(* CODESYS project TrafficLight.project

Project tree, tasks and I/O mapping:
  Device : Elmo Platinum Maestro, Elmo Motion Control, version 1.0.0.2
    application Application
      libraries: Standard, * (System); VisuDialogs, * (System)
      task MainTask (cyclic, interval t#20ms, priority 1) calls PLC_PRG
      task VISU_TASK (cyclic, interval 100 ms, priority 31) calls VisuElems.Visu_Prg
      program PLC_PRG [ST]
      visualisation Visualization
      Structure/
        data type stCarX
        data type stCarY
      function block fbModeSwitch [ST]
      function fTimetoString [ST]
      function block fbGreenTimeCondition [ST]
      function block fbYellowTimeCondition [ST]
      function block fbClearTimeCondition [ST]
      function block fbFrontandBackCar [ST]
    Elmo_Master_Device : Elmo Master Device, Elmo, version 1.0.0.2
  libraries: VisuSymbols, 3.5.10.0 (System)
  text list GlobalTextList
*)

// Device/Application/Structure/stCarX
TYPE stCarX :
STRUCT
	iMove_x: INT;
	//iBase_x: ARRAY[1..5] OF INT := [243,195,157,113,69];
	//iBase_x: ARRAY[1..5] OF INT;
END_STRUCT
END_TYPE

// Device/Application/Structure/stCarY
TYPE stCarY :
STRUCT
	iMove_y: INT;
	//iBase_y: ARRAY[1..5] OF INT;
END_STRUCT
END_TYPE

// Device/Application/PLC_PRG
PROGRAM PLC_PRG
VAR CONSTANT
	c_dwRoadColor : DWORD := 16#88888888;
	c_dwLaneColor: DWORD := 16#FFFFFF00;
	c_dwTLbg: DWORD := 16#88000000;
END_VAR
VAR
	xPush: BOOL;
	tonTimer1: ton;
	tonTimer2: ton;
	tonTimer3: ton;
	xStart1: BOOL;
	xStart2: BOOL;
	xStart3: BOOL;
	uiTrafficSig: UINT:=0;
	
	xGreen1 : BOOL;
	xYellow1 : BOOL;
	xRed1 : BOOL;
	xRed2 : BOOL;
	xYellow2 : BOOL;
	xGreen2 : BOOL;
	tTimer1: TIME := T#7000MS;
	tTimer2: TIME := T#5000MS;
	tTimer3: TIME := T#4000MS;
	
	tSTime1: STRING := 'T#7s';
	tSTime2: STRING := 'T#5s';
	tSTime3: STRING := 'T#4s';
	
	tSeTime1: STRING := 'T#7s';
	tSeTime2: STRING := 'T#5s';
	tSeTime3: STRING := 'T#4s';
	tRed : STRING;
	
	tEditTime1 : TIME := T#7000MS;
	tEditTime2 : TIME := T#5000MS;
	tEditTime3 : TIME := T#4000MS;
	sEditTime1 : STRING;
	sEditTime2 : STRING;
	sEditTime3 : STRING;
	
	stCarX: ARRAY [1..5] OF stCarX;
	uiLoop: UINT;
	
	iBase_x : ARRAY[1..5] OF INT := [250,200,150,100,50];
		
	stCarY: ARRAY [1..5] OF stCarY;
	uiLoop2: UINT;
	iBase_y : ARRAY[1..5] OF INT := [450,500,550,600,650];
	
	iMoveUser1X: INT;
	iMoveUser1Y: INT;
	iMoveUser2X: INT;
	iMoveUser2Y: INT;
	iMoveUser1Z: INT;
	iMoveUser2Z: INT;
	
	iCurrent: INT;
	iCurrent2: INT;
	iForward: INT;
	iForward2: INT;
	iBack: INT;
	iBack2: INT;
    sMode: STRING;
	iTemp: INT;
	iTemp2: INT;
	iStart: INT;
	iStart2: INT;
	
	fbMode : fbModeSwitch;
	fbGreenTime: fbGreenTimeCondition;
	fbYellowTime: fbYellowTimeCondition;
	fbClearTime: fbClearTimeCondition;
	fbFrontBack: fbFrontandBackCar;
END_VAR

//Mode Switch
fbMode(ix_Push := xPush,os_Mode => sMode);

//Time Edit
tSTime1 := fTimetoString(it_Time := tTimer1);
tSTime2 := fTimetoString(it_Time := tTimer2);
tSTime3 := fTimetoString(it_Time := tTimer3);
tSeTime1 := fTimetoString(it_Time := tEditTime1);
tSeTime2 := fTimetoString(it_Time := tEditTime2);
tSeTime3 := fTimetoString(it_Time := tEditTime3);

//Green Time Edit Conditions
fbGreenTime(it_EditTime1 := tEditTime1 ,it_Timer2 := tTimer2 ,it_Timer3 := tTimer3 ,ot_timer1 => tTimer1 ,os_EditTime1 => sEditTime1);
//Yellow Time Edit Conditions
fbYellowTime(it_EditTime2 := tEditTime2 ,it_EditTime1 := tEditTime1 ,it_EditTime3 := tEditTime3 ,ot_timer2 => tTimer2 ,os_EditTime2 => sEditTime2);
//Clear Time Edit Conditions
fbClearTime(it_EditTime3 := tEditTime3 ,it_EditTime1 := tEditTime1 ,it_EditTime2 := tEditTime2 ,ot_timer3 => tTimer3 ,os_EditTime3 => sEditTime3);

//Traffic Light Sequence
CASE uiTrafficSig OF
	0:
	     xRed1 := FALSE;
	     xGreen1 := TRUE;
	     xRed2 := TRUE;
	     tonTimer1(IN := xStart1, PT := tTimer1);
	     xStart1 := TRUE;
	     IF tonTimer1.Q = TRUE THEN
		   xStart1 := FALSE;
		   xGreen1 := FALSE;
		   uiTrafficSig := 10;
	     END_IF
	10:
	   tonTimer2(IN := xStart2, PT := tTimer2);
	   xStart2 := TRUE;
	   xYellow1 := TRUE;
	   IF tonTimer2.Q = TRUE THEN
		   xStart2 := FALSE;
		   //xYellow1 := FALSE;
		   uiTrafficSig := 20;
	   END_IF
	20:
	   tonTimer3(IN := xStart3, PT := tTimer3);
	   xStart3 := TRUE;
	   xYellow1 := FALSE;
	   xRed1 := TRUE;
	   IF tonTimer3.Q = TRUE THEN
		   xStart3 := FALSE;
		   IF xPush = TRUE THEN
			   uiTrafficSig := 60;
		   ELSE
			   uiTrafficSig := 30;
		   END_IF
	   END_IF
	30:
	       xRed2 := FALSE;
	       xGreen2 := TRUE;
	       tonTimer1(IN := xStart1, PT := tTimer1);
	       xStart1 := TRUE;
	       IF tonTimer1.Q = TRUE THEN
			   xStart1 := FALSE;
			   xGreen2 := FALSE;
			   uiTrafficSig := 40;
	       END_IF
	40:
	   xYellow2 := TRUE;
	   tonTimer2(IN := xStart2, PT := tTimer2);
	   xStart2 := TRUE;
	   IF tonTimer2.Q = TRUE THEN
		   xStart2 := FALSE;
		   //xYellow2 := FALSE;
		   uiTrafficSig := 50;
	   END_IF
	50:
	   xYellow2 := FALSE;
	   xRed2 := TRUE;
	   tonTimer3(IN := xStart3, PT := tTimer3);
	   xStart3 := TRUE;
	   IF tonTimer3.Q = TRUE THEN
		   xStart3 := FALSE;
		   IF xPush = TRUE THEN
			   uiTrafficSig := 60;
		   ELSE
			   uiTrafficSig := 0;
		   END_IF
	   END_IF
	60:
	IF xPush = TRUE THEN
	   xRed1 := TRUE;
	   xRed2 := TRUE;
	   xYellow1 := FALSE;
	   xYellow2 := FALSE;
	   xGreen1 := FALSE;
	   xGreen2 := FALSE;
	ELSE
		uiTrafficSig := 0;
	END_IF
END_CASE

//Red Time Total
tRed := fTimetoString(it_Time := tTimer1 + tTimer2 + tTimer3);

FOR uiLoop:=1 TO 5 BY 1 DO
	iCurrent := iBase_x[uiLoop] + stCarX[uiLoop].iMove_x;
	
    IF xGreen1 = TRUE OR xYellow1 = TRUE THEN
		iTemp := 0;
		FOR uiLoop2:=1 TO 5 BY 1 DO
			//knowing front and back cars of each
			fbFrontBack(iui_Loop:=uiLoop,ii_Base_x:=iBase_x,stCarX:=stCarX,oi_Forward => iForward, oi_Back => iBack);
			
			//condition 1 for stopping at green signal if any opposite cars are seen at intersection
			IF iBase_y[uiLoop2] + stCarY[uiLoop2].iMove_y < 450 AND iBase_y[uiLoop2] + stCarY[uiLoop2].iMove_y > 175 THEN
				stCarX[uiLoop].iMove_x := stCarX[uiLoop].iMove_x +0;
				iTemp := 0;
			ELSE
					IF iBase_y[uiLoop2] + stCarY[uiLoop2].iMove_y > 450 OR iBase_y[uiLoop2] + stCarY[uiLoop2].iMove_y < 175 THEN
						iTemp := iTemp + 1;
					END_IF
				
			END_IF
		END_FOR
		
		//condition 2 for stopping at green signal if any opposite cars are seen at intersection
		IF iCurrent >= 425 AND iCurrent < 450 AND iTemp < 5 THEN
			stCarX[uiLoop].iMove_x := stCarX[uiLoop].iMove_x +0;
			IF uiLoop = 5 THEN
					stCarX[1].iMove_x := stCarX[1].iMove_x + 0;
			ELSE
					stCarX[uiLoop + 1].iMove_x := stCarX[uiLoop + 1].iMove_x + 0;
			END_IF
		END_IF
		
		//Condition for car movement at green signal and also condition for reverse
		IF (iTemp >= 4 OR (iCurrent < 425 AND iForward - iCurrent > 50 AND iForward > iCurrent) OR (iCurrent > 450) OR (iCurrent < 425 AND iCurrent - iForward > 50 AND iCurrent > iForward)) THEN
			IF stCarX[uiLoop].iMove_x <= -500 THEN
				IF iStart >= 5 THEN
					stCarX[uiLoop].iMove_x := stCarX[uiLoop].iMove_x +1;
				ELSE
					stCarX[uiLoop].iMove_x := stCarX[uiLoop].iMove_x +0;
				END_IF
			ELSE
				stCarX[uiLoop].iMove_x := stCarX[uiLoop].iMove_x +1;
			END_IF
		END_IF
		
	ELSIF xRed1 = TRUE THEN
		iTemp:= 0;
		iCurrent := iBase_x[uiLoop] + stCarX[uiLoop].iMove_x;

		fbFrontBack(iui_Loop:=uiLoop,ii_Base_x:=iBase_x,stCarX:=stCarX,oi_Forward => iForward, oi_Back => iBack);
			//Movement Condition 1 and reverse condition during red light
			IF iCurrent < 425 AND iForward - iCurrent > 50 AND iForward > iCurrent THEN
				IF stCarX[uiLoop].iMove_x <= -500 THEN
				 IF iStart >= 5 THEN
					stCarX[uiLoop].iMove_x := stCarX[uiLoop].iMove_x +1;
				 ELSE
					stCarX[uiLoop].iMove_x := stCarX[uiLoop].iMove_x +0;
				 END_IF
			  ELSE
				stCarX[uiLoop].iMove_x := stCarX[uiLoop].iMove_x +1;
			END_IF
				
			//Movement Condition 2 and reverse condition during red light
			ELSIF iCurrent < 425 AND iForward < 425 AND iCurrent - iForward > 50 THEN
				IF stCarX[uiLoop].iMove_x <= -500 THEN
				 IF iStart >= 5 THEN
					stCarX[uiLoop].iMove_x := stCarX[uiLoop].iMove_x +1;
				 ELSE
					stCarX[uiLoop].iMove_x := stCarX[uiLoop].iMove_x +0;
				 END_IF
			   ELSE
				stCarX[uiLoop].iMove_x := stCarX[uiLoop].iMove_x +1;
			  END_IF
			
          //Stop Condition 1	
		  ELSIF iCurrent < 425 THEN
			  stCarX[uiLoop].iMove_x := stCarX[uiLoop].iMove_x + 0;
		  //Intersection Speeding Condition
		  ELSIF iCurrent > 425 AND iCurrent < 800 THEN
			  stCarX[uiLoop].iMove_x := stCarX[uiLoop].iMove_x + 5;
			
          //Movement Condition 3	
		  ELSIF iCurrent >= 800 THEN
			  stCarX[uiLoop].iMove_x := stCarX[uiLoop].iMove_x + 5;
			  
			END_IF
			
	END_IF
		
	//Condition at end
	IF iBase_x[uiLoop] + stCarX[uiLoop].iMove_x >= 1900 THEN
		fbFrontBack(iui_Loop:=uiLoop,ii_Base_x:=iBase_x,stCarX:=stCarX,oi_Forward => iForward, oi_Back => iBack);
		
		IF(iStart >= 5)THEN
			iStart := 0;
		END_IF
		stCarX[uiLoop].iMove_x := -500;
		iStart := iStart + 1;
    END_IF
	
END_FOR

FOR uiLoop2:=1 TO 5 BY 1 DO
	
	iCurrent2 := iBase_y[uiLoop2] + stCarY[uiLoop2].iMove_y;
	
	IF xGreen2 = TRUE OR xYellow2 = TRUE THEN
		iTemp2 := 0;
		FOR uiLoop:=1 TO 5 BY 1 DO
			IF uiLoop2 = 1 THEN
				iForward2 := iBase_y[5] + stCarY[5].iMove_y;
			    iBack2 := iBase_y[uiLoop2 + 1] + stCarY[uiLoop2 + 1].iMove_y;
			ELSIF uiLoop2 = 5 THEN
				iForward2 := iBase_y[uiLoop2 - 1] + stCarY[uiLoop2 - 1].iMove_y;
			    iBack2 := iBase_y[1] + stCarY[1].iMove_y;
			ELSE
				iForward2 := iBase_y[uiLoop2 - 1] + stCarY[uiLoop2 - 1].iMove_y;
			    iBack2 := iBase_y[uiLoop2 + 1] + stCarY[uiLoop2 + 1].iMove_y;
			END_IF
			//condition 1 for stopping at green signal if any opposite cars are seen at intersection
			IF iBase_x[uiLoop] + stCarX[uiLoop].iMove_x > 425 AND iBase_x[uiLoop] + stCarX[uiLoop].iMove_x < 800 THEN
				stCarX[uiLoop].iMove_x := stCarX[uiLoop].iMove_x +0;
				iTemp2 := 0;
			ELSE
					IF iBase_x[uiLoop] + stCarX[uiLoop].iMove_x < 425 OR iBase_x[uiLoop] + stCarX[uiLoop].iMove_x > 800 THEN
						iTemp2 := iTemp2 + 1;
					END_IF
				
			END_IF
		END_FOR
		
		//condition 2 for stopping at green signal if any opposite cars are seen at intersection
		IF iCurrent2 <= 450 AND iCurrent2 > 425 AND iTemp2 < 5 THEN
			stCarY[uiLoop2].iMove_y := stCarY[uiLoop2].iMove_y +0;
			IF uiLoop2 = 5 THEN
					stCarY[1].iMove_y := stCarY[1].iMove_y + 0;
			ELSE
					stCarY[uiLoop2 + 1].iMove_y := stCarY[uiLoop2 + 1].iMove_y + 0;
			END_IF
		END_IF
		//Condition for car movement at green signal and also condition for reverse
		IF iTemp2 >= 4 OR (iCurrent2 > 450 AND iCurrent2 - iForward2 > 50 AND iForward2 < iCurrent2) OR (iCurrent2 < 425) OR (iCurrent2 > 450 AND iForward2 - iCurrent2 > 50 AND iCurrent2 < iForward2)THEN
			IF stCarY[uiLoop2].iMove_y >= 1050 THEN
				IF iStart2 >= 5 THEN
					stCarY[uiLoop2].iMove_y := stCarY[uiLoop2].iMove_y -1;
				ELSE
					stCarY[uiLoop2].iMove_y := stCarY[uiLoop2].iMove_y +0;
				END_IF
			ELSE
				stCarY[uiLoop2].iMove_y := stCarY[uiLoop2].iMove_y -1;
			END_IF
		END_IF
		
		
	ELSIF xRed2 = TRUE THEN
		iCurrent2 := iBase_y[uiLoop2] + stCarY[uiLoop2].iMove_y;
		iTemp2 := 0;
		
			IF uiLoop2 = 1 THEN
				iForward2 := iBase_y[5] + stCarY[5].iMove_y;
			    iBack2 := iBase_y[uiLoop2 + 1] + stCarY[uiLoop2 + 1].iMove_y;
			ELSIF uiLoop2 = 5 THEN
				iForward2 := iBase_y[uiLoop2 - 1] + stCarY[uiLoop2 - 1].iMove_y;
			    iBack2 := iBase_y[1] + stCarY[1].iMove_y;
			ELSE
				iForward2 := iBase_y[uiLoop2 - 1] + stCarY[uiLoop2 - 1].iMove_y;
			    iBack2 := iBase_y[uiLoop2 + 1] + stCarY[uiLoop2 + 1].iMove_y;
			END_IF
			//Movement Condition 1 and reverse condition during red light
			IF iCurrent2 > 450 AND  iCurrent2 - iForward2 > 50 AND iForward2 < iCurrent2 THEN
				IF stCarY[uiLoop2].iMove_y >= 1050 THEN
				 IF iStart2 >= 5 THEN
					stCarY[uiLoop2].iMove_y := stCarY[uiLoop2].iMove_y -1;
				 ELSE
					stCarY[uiLoop2].iMove_y := stCarY[uiLoop2].iMove_y +0;
				 END_IF
			   ELSE
				stCarY[uiLoop2].iMove_y := stCarY[uiLoop2].iMove_y -1;
			   END_IF
			   //Movement Condition 2 and reverse condition during red light
			ELSIF iCurrent2 > 450 AND iForward2 > 450 AND  iForward2 - iCurrent2 > 50 THEN
				IF stCarY[uiLoop2].iMove_y >= 1050 THEN
				 IF iStart2 >= 5 THEN
					stCarY[uiLoop2].iMove_y := stCarY[uiLoop2].iMove_y -1;
				 ELSE
					stCarY[uiLoop2].iMove_y := stCarY[uiLoop2].iMove_y +0;
				 END_IF
			   ELSE
				stCarY[uiLoop2].iMove_y := stCarY[uiLoop2].iMove_y -1;
			   END_IF
			   //Stop Condition 1
			ELSIF iCurrent2 > 450 THEN
			  stCarY[uiLoop2].iMove_y := stCarY[uiLoop2].iMove_y + 0;
			  //Intersection Speeding Condition
			ELSIF iCurrent2 < 450 AND iCurrent2 > 175 THEN
			    stCarY[uiLoop2].iMove_Y := stCarY[uiLoop2].iMove_y - 5;
				
				//Movement Condition 3
		    ELSIF iCurrent2 <= 175 THEN
			  stCarY[uiLoop2].iMove_y := stCarY[uiLoop2].iMove_y - 5;
			  
			END_IF
			
	END_IF
		
		//Condition at end
	IF iBase_y[uiLoop2] + stCarY[uiLoop2].iMove_y <= -100 THEN
		IF uiLoop2 = 1 THEN
				iForward2 := iBase_y[5] + stCarY[5].iMove_y;
			    iBack2 := iBase_y[uiLoop2 + 1] + stCarY[uiLoop2 + 1].iMove_y;
		ELSIF uiLoop = 5 THEN
				iForward2 := iBase_y[uiLoop2 - 1] + stCarY[uiLoop2 - 1].iMove_y;
			    iBack2 := iBase_y[1] + stCarY[1].iMove_y;
		ELSE
				iForward2 := iBase_y[uiLoop2 - 1] + stCarY[uiLoop2 - 1].iMove_y;
			    iBack2 := iBase_y[uiLoop2 + 1] + stCarY[uiLoop2 + 1].iMove_y;
		END_IF
			IF(iStart2 >= 5)THEN
			  iStart2 := 0;
		    END_IF
		    stCarY[uiLoop2].iMove_y := 1050;
		    iStart2 := iStart2 + 1;
    END_IF
	
END_FOR

//People Movement at crossing
CASE iMoveUser1Z OF
	0:
	   IF xGreen1 = TRUE THEN
		   iMoveUser1X := iMoveUser1X + 5;
	       IF iMoveUser1X = 250 THEN
	         iMoveUser1Z:= 250;
	       END_IF
	   END_IF
	   
	250:
	   IF xGreen2 = TRUE THEN
		   iMoveUser1Y := iMoveUser1Y - 5;
		   IF iMoveUser1Y = -175 THEN
	         iMoveUser1Z:= 500;
	       END_IF
	   END_IF
	   
	500:
	   IF xGreen1 = TRUE THEN
		   iMoveUser1X := iMoveUser1X - 5;
	       IF iMoveUser1X = 0 THEN
	         iMoveUser1Z:= 750;
	       END_IF
	   END_IF
	   
	 750:
	   IF xGreen2 = TRUE THEN
		   iMoveUser1Y := iMoveUser1Y + 5;
		   IF iMoveUser1Y = 0 THEN
	         iMoveUser1Z:= 0;
	       END_IF
	   END_IF
		
END_CASE


CASE iMoveUser2Z OF
	0:
	   IF xGreen1 = TRUE THEN
		   iMoveUser2X := iMoveUser2X - 5;
	       IF iMoveUser2X = -225 THEN
	         iMoveUser2Z:= 250;
	       END_IF
	   END_IF
	   
	250:
	   IF xGreen2 = TRUE THEN
		   iMoveUser2Y := iMoveUser2Y + 5;
		   IF iMoveUser2Y = 175 THEN
	         iMoveUser2Z:= 500;
	       END_IF
	   END_IF
	   
	500:
	   IF xGreen1 = TRUE THEN
		   iMoveUser2X := iMoveUser2X + 5;
	       IF iMoveUser2X = 0 THEN
	         iMoveUser2Z:= 750;
	       END_IF
	   END_IF
	   
	 750:
	   IF xGreen2 = TRUE THEN
		   iMoveUser2Y := iMoveUser2Y - 5;
		   IF iMoveUser2Y = 0 THEN
	         iMoveUser2Z:= 0;
	       END_IF
	   END_IF
		
END_CASE

END_PROGRAM

// Device/Application/fTimetoString
FUNCTION fTimetoString : STRING
VAR_INPUT
	it_Time: TIME;
END_VAR
VAR
END_VAR

fTimetoString := TIME_TO_STRING(it_Time);

END_FUNCTION

// Device/Application/fbModeSwitch
FUNCTION_BLOCK fbModeSwitch
VAR_INPUT
	ix_Push: BOOL;
END_VAR
VAR_OUTPUT
	os_Mode: STRING;
END_VAR
VAR
END_VAR

IF ix_Push = TRUE THEN
	os_Mode := 'STOP';
ELSE
	os_Mode := 'AUTO';
END_IF

END_FUNCTION_BLOCK

// Device/Application/fbGreenTimeCondition
FUNCTION_BLOCK fbGreenTimeCondition
VAR_INPUT
	it_EditTime1: TIME;
	it_Timer2: TIME;
	it_Timer3: TIME;
END_VAR
VAR_OUTPUT
	ot_Timer1: TIME;
	os_EditTime1: STRING;
END_VAR
VAR
END_VAR

IF it_EditTime1 >= T#7000MS AND it_EditTime1 > it_Timer2 AND it_EditTime1 > it_Timer3 AND it_EditTime1 <= T#30000MS THEN
			 ot_Timer1 := it_EditTime1;
			 os_EditTime1 := 'Valid';
ELSE
	os_EditTime1 := 'Invalid';
END_IF

END_FUNCTION_BLOCK

// Device/Application/fbYellowTimeCondition
FUNCTION_BLOCK fbYellowTimeCondition
VAR_INPUT
	it_EditTime2: TIME;
	it_EditTime1: TIME;
	it_EditTime3: TIME;
END_VAR
VAR_OUTPUT
	ot_Timer2: TIME;
	os_EditTime2: STRING;
END_VAR
VAR
END_VAR

IF it_EditTime2 >= T#5000MS AND it_EditTime2 < it_EditTime1 AND it_EditTime2 > it_EditTime3 AND it_EditTime2 <= T#28000MS THEN
			 ot_Timer2 := it_EditTime2;
			 os_EditTime2 := 'Valid';
ELSE
	os_EditTime2 := 'Invalid';
END_IF

END_FUNCTION_BLOCK

// Device/Application/fbClearTimeCondition
FUNCTION_BLOCK fbClearTimeCondition
VAR_INPUT
	it_EditTime3: TIME;
	it_EditTime1: TIME;
	it_EditTime2: TIME;
END_VAR
VAR_OUTPUT
	ot_Timer3: TIME;
	os_EditTime3: STRING;
END_VAR
VAR
END_VAR

IF it_EditTime3 >= T#4000MS AND it_EditTime3 < it_EditTime1 AND it_EditTime3 < it_EditTime2 AND it_EditTime3 <= T#27000MS THEN
			 ot_Timer3 := it_EditTime3;
			 os_EditTime3 := 'Valid';
ELSE
	os_EditTime3 := 'Invalid';
END_IF

END_FUNCTION_BLOCK

// Device/Application/fbFrontandBackCar
FUNCTION_BLOCK fbFrontandBackCar
VAR_INPUT
	iui_Loop: UINT;
	ii_Base_x : ARRAY[1..5] OF INT := [250,200,150,100,50];
	stCarX: ARRAY [1..5] OF stCarX;
END_VAR
VAR_OUTPUT
	oi_Forward: INT;
	oi_Back: INT;
END_VAR
VAR
END_VAR

IF iui_Loop = 1 THEN
		oi_Forward := ii_Base_x[5] + stCarX[5].iMove_x;
	    oi_Back := ii_Base_x[iui_Loop + 1] + stCarX[iui_Loop + 1].iMove_x;
ELSIF iui_Loop = 5 THEN
		oi_Forward := ii_Base_x[iui_Loop - 1] + stCarX[iui_Loop - 1].iMove_x;
		oi_Back := ii_Base_x[1] + stCarX[1].iMove_x;
ELSE
		oi_Forward := ii_Base_x[iui_Loop - 1] + stCarX[iui_Loop - 1].iMove_x;
	    oi_Back := ii_Base_x[iui_Loop + 1] + stCarX[iui_Loop + 1].iMove_x;
END_IF

END_FUNCTION_BLOCK

// Device/Application/Visualization
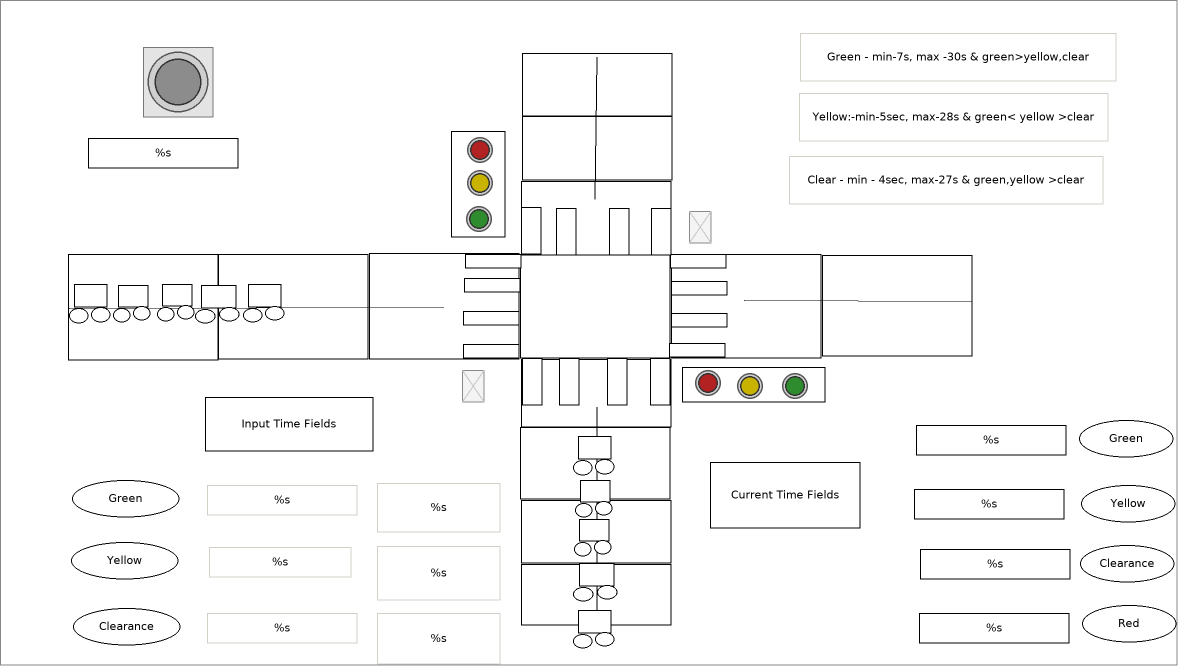
VISUALIZATION Visualization  // 1178x666
    Rectangle (68,254 150x106), colour variable: PLC_PRG.c_dwRoadColor
    Rectangle (218,254 150x105), colour variable: PLC_PRG.c_dwRoadColor
    Rectangle (369,253 150x106), colour variable: PLC_PRG.c_dwRoadColor
    Rectangle (520,254 150x104), colour variable: PLC_PRG.c_dwRoadColor
    Rectangle (671,254 150x104), colour variable: PLC_PRG.c_dwRoadColor
    Rectangle (822,255 150x101), colour variable: PLC_PRG.c_dwRoadColor
    Rectangle (521,181 150x74), colour variable: PLC_PRG.c_dwRoadColor
    Rectangle (522,116 150x64), colour variable: PLC_PRG.c_dwRoadColor
    Rectangle (522,53 150x63), colour variable: PLC_PRG.c_dwRoadColor
    Rectangle (521,359 150x68), colour variable: PLC_PRG.c_dwRoadColor
    Rectangle (520,427 150x72), colour variable: PLC_PRG.c_dwRoadColor
    Rectangle (521,500 150x63), colour variable: PLC_PRG.c_dwRoadColor
    Rectangle (521,564 150x61), colour variable: PLC_PRG.c_dwRoadColor
    Line (69,308) (443,307)
        p2175578022: PLC_PRG.c_dwLaneColor
    Line (744,300) (972,301)
        p2175578022: PLC_PRG.c_dwLaneColor
    Line (595,199) (597,57)
        p2175578022: PLC_PRG.c_dwLaneColor
    Line (597,623) (597,407)
        p2175578022: PLC_PRG.c_dwLaneColor
    Rectangle (463,344 56x14)
    Rectangle (463,311 56x14)
    Rectangle (464,278 56x14)
    Rectangle (465,254 56x14)
    Rectangle (670,254 56x14)
    Rectangle (671,281 56x14)
    Rectangle (671,313 56x14)
    Rectangle (669,343 56x14)
    Rectangle (521,207 20x47)
    Rectangle (556,208 20x47)
    Rectangle (609,208 20x47)
    Rectangle (651,208 20x47)
    Rectangle (522,358 20x47)
    Rectangle (559,358 20x47)
    Rectangle (607,358 20x47)
    Rectangle (650,358 20x47)
    Rectangle (451,131 54x106), colour variable: PLC_PRG.c_dwTLbg
    Rectangle (682,367 143x35), colour variable: PLC_PRG.c_dwTLbg
    Lamp1 (465,135 30x30), variable: PLC_PRG.xRed1, style: Lamp-Lamp1-Red
    Lamp1 (465,168 30x30), variable: PLC_PRG.xYellow1, style: Lamp-Lamp1-Yellow
    Lamp1 (464,204 30x30), variable: PLC_PRG.xGreen1, style: Lamp-Lamp1-Green
    Lamp1 (693,368 30x30), variable: PLC_PRG.xRed2, style: Lamp-Lamp1-Red
    Lamp1 (735,371 30x30), variable: PLC_PRG.xYellow2, style: Lamp-Lamp1-Yellow
    Lamp1 (780,371 30x30), variable: PLC_PRG.xGreen2, style: Lamp-Lamp1-Green
    PushSwitchLed (143,47 70x70), variable: PLC_PRG.xPush, behaviour: TOGGLE, style: Switch-PushSwitchLed-Gray
    Group (243,284 41x38)
        p3560616238: PLC_PRG.stCarX[1].iMove_x
        RoundedRectangle (5,0 33x23), colour variable: 16#FF0000FF
        Ellipse (0,24 19x14)
        Ellipse (22,22 19x14)
    Group (195,285 44x38)
        p3560616238: PLC_PRG.stCarX[2].iMove_x
        RoundedRectangle (6,0 35x23), colour variable: 16#FF0000FF
        Ellipse (0,24 20x14)
        Ellipse (24,22 20x14)
    Group (157,284 37x37)
        p3560616238: PLC_PRG.stCarX[3].iMove_x
        RoundedRectangle (5,0 30x22), colour variable: 16#FFFF0000
        Ellipse (0,23 17x14)
        Ellipse (20,21 17x14)
    Group (69,284 41x39)
        p3560616238: PLC_PRG.stCarX[5].iMove_x
        RoundedRectangle (5,0 33x23), colour variable: 16#FF00FF00
        Ellipse (0,24 19x15)
        Ellipse (22,23 19x15)
    Group (113,285 37x37)
        p3560616238: PLC_PRG.stCarX[4].iMove_x
        RoundedRectangle (5,0 30x22), colour variable: 16#FFFFFF00
        Ellipse (0,23 17x14)
        Ellipse (20,21 17x14)
    Group (573,436 41x39)
        p2738717112: PLC_PRG.stCarY[1].iMove_y
        RoundedRectangle (5,0 33x23), colour variable: 16#FF00FF00
        Ellipse (0,24 19x15)
        Ellipse (22,23 19x15)
    Group (573,610 41x38)
        p2738717112: PLC_PRG.stCarY[5].iMove_y
        RoundedRectangle (5,0 33x23), colour variable: 16#FF0000FF
        Ellipse (0,24 19x14)
        Ellipse (22,22 19x14)
    Group (573,563 44x38)
        p2738717112: PLC_PRG.stCarY[4].iMove_y
        RoundedRectangle (6,0 35x23), colour variable: 16#FF0000FF
        Ellipse (0,24 20x14)
        Ellipse (24,22 20x14)
    Group (574,519 37x37)
        p2738717112: PLC_PRG.stCarY[3].iMove_y
        RoundedRectangle (5,0 30x22), colour variable: 16#FFFF0000
        Ellipse (0,23 17x14)
        Ellipse (20,21 17x14)
    Group (575,480 37x37)
        p2738717112: PLC_PRG.stCarY[2].iMove_y
        RoundedRectangle (5,0 30x22), colour variable: 16#FFFFFF00
        Ellipse (0,23 17x14)
        Ellipse (20,21 17x14)
    Image (462,370 22x32), image: VisuSymbols.Symbols.AddUser
        p3560616238: PLC_PRG.iMoveUser1X
        p2738717112: PLC_PRG.iMoveUser1Y
    Image (689,211 22x32), image: VisuSymbols.Symbols.AddUser
        p3560616238: PLC_PRG.iMoveUser2X
        p2738717112: PLC_PRG.iMoveUser2Y
    RoundedRectangle (88,138 150x30), "%s", text variable: PLC_PRG.sMode
    Textfield (207,485 150x30), "%s", text variable: PLC_PRG.tSeTime1
        OnMouseClick: write PLC_PRG.tEditTime1 via Default
    Rectangle (916,425 150x30), "%s", text variable: PLC_PRG.tSTime1
        OnMouseClick: write PLC_PRG.tTimer1 via Default
    Textfield (209,547 142x30), "%s", text variable: PLC_PRG.tSeTime2
        OnMouseClick: write PLC_PRG.tEditTime2 via Default
    Textfield (207,613 150x30), "%s", text variable: PLC_PRG.tSeTime3
        OnMouseClick: write PLC_PRG.tEditTime3 via Default
    Rectangle (205,397 168x54), "Input Time Fields"
    Ellipse (72,480 107x37), "Green"
    Ellipse (71,542 107x37), "Yellow"
    Ellipse (73,608 107x37), "Clearance"
    Rectangle (914,489 150x30), "%s", text variable: PLC_PRG.tSTime2
        OnMouseClick: write PLC_PRG.tTimer2 via Default
    Rectangle (920,549 150x30), "%s", text variable: PLC_PRG.tSTime3
        OnMouseClick: write PLC_PRG.tTimer3 via Default
    Rectangle (919,613 150x30), "%s", text variable: PLC_PRG.tRed
    RoundedRectangle (710,462 150x66), "Current Time Fields"
    Ellipse (1079,420 94x37), "Green"
    Ellipse (1081,485 94x37), "Yellow"
    Ellipse (1080,545 94x37), "Clearance"
    Ellipse (1082,605 94x37), "Red"
    Textfield (377,483 123x49), "%s", text variable: PLC_PRG.sEditTime1
    Textfield (377,546 123x54), "%s", text variable: PLC_PRG.sEditTime2
    Textfield (377,613 123x51), "%s", text variable: PLC_PRG.sEditTime3
    Textfield (800,33 316x48), "Green - min-7s, max -30s & green>yellow,clear"
    Textfield (799,93 309x48), "Yellow:-min-5sec, max-28s & green< yellow >clear"
    Textfield (789,156 314x48), "Clear - min - 4sec, max-27s & green,yellow >clear"
END_VISUALIZATION
